{attribute 'no_explicit_call' := 'do not call this FB directly'}{attribute 'enable_dynamic_creation'}
FUNCTION_BLOCK FINAL Node_Literal_BOOL EXTENDS Node
VAR
	value : _BOOL(FALSE);
	out : _BOOL(FALSE);
END_VAR

METHOD PUBLIC Clone : I_Node
VAR
	pointerToNode : POINTER TO Node_Literal_BOOL;
END_VAR
pointerToNode := __NEW(Node_Literal_BOOL);
Clone := pointerToNode^;
END_METHOD

METHOD FB_init : BOOL
VAR_INPUT
	bInitRetains : BOOL; // if TRUE, the retain variables are initialized (warm start / cold start)
	bInCopyCode : BOOL;  // if TRUE, the instance afterwards gets moved into the copy code (online change)
END_VAR
Parameters.AddDataAsParameter('value', value);
OutputPorts.AddDataAsOutputPort('out', out);
END_METHOD

METHOD PROTECTED OnExecute : HRESULT
VAR
END_VAR
out.value := value.value;
END_METHOD

END_FUNCTION_BLOCK

(* stored: Version 1.1.0.1, ProductVersion 3.1.4024.12
   POU Node_Literal_BOOL: Id {12053a2d-1811-05b8-274f-6b729ca726b1}, SpecialFunc None
   Folder Constructor: Id {066907f7-a45f-41f8-bd90-26a3e7745138}
   Method Clone: Id {2952cb38-91f7-44e6-a935-c5279debf1b1}
   Method FB_init: Id {2b84cc63-8aa0-4cfa-9150-5d2446c77c1a}
   Method OnExecute: Id {17896f32-d471-0aa9-3949-762ff3592dce} *)
